TYPE ST_StepCriterionResult : STRUCT
    (* 被评估的 CFF 步骤。 *)
    eStep : E_CffStep;
    (* 实际步骤结束原因。 *)
    eEndCause : E_StepEndCause;
    (* 主判据是否已经锁存。 *)
    bPrimaryLatched : BOOL;
    (* 次级判据是否已经锁存。 *)
    bSecondaryLatched : BOOL;
    (* 步骤是否判为不合格。 *)
    bNok : BOOL;
    (* 判据触发时的周期计数。 *)
    nTriggerCycle : UDINT;
    (* 步骤是否过短。 *)
    bTooShort : BOOL;
    (* 合格力带保持时间是否满足。 *)
    bQualifiedForceHoldMet : BOOL;
    (* 合格力带实际保持时间，单位秒。 *)
    rQualifiedForceHoldTime_s : LREAL;
    (* 锁存的轴向力，单位千牛。 *)
    rLatchedForce_kN : LREAL;
    (* 锁存的相对位置，单位毫米。 *)
    rLatchedRelativePosition_mm : LREAL;
    (* 锁存的步骤时间，单位秒。 *)
    rLatchedStepTime_s : LREAL;
END_STRUCT
END_TYPE

(* stored: Version 1.1.0.1
   DUT ST_StepCriterionResult: Id {D3100000-0000-4000-8000-000000000017} *)
